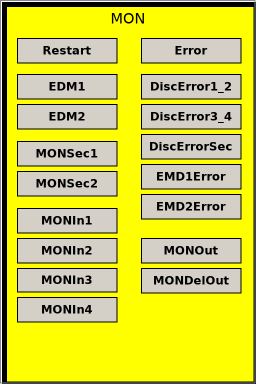
VISUALIZATION V_PH_MON  // 256x384
VAR_INPUT
	stSafetyMon				: ST_SAFETY_FBMON;
	
END_VAR
    Rectangle (2,2 256x384), colour toggle: stSafetyMon.bGeneralError
    Label (5,6 246x25), "MON"
    RoundedRectangle (17,38 100x25), "Restart", colour toggle: stSafetyMon.uStatus.stStatusWords.wInputs.0
    RoundedRectangle (17,74 100x25), "EDM1", colour toggle: stSafetyMon.uStatus.stStatusWords.wInputs.1
    RoundedRectangle (17,297 100x25), "MONIn4", colour toggle: stSafetyMon.uStatus.stStatusWords.wInputs.11
    RoundedRectangle (17,104 100x25), "EDM2", colour toggle: stSafetyMon.uStatus.stStatusWords.wInputs.2
    RoundedRectangle (17,171 100x25), "MONSec2", colour toggle: stSafetyMon.uStatus.stStatusWords.wInputs.4
    RoundedRectangle (17,268 100x24), "MONIn3", colour toggle: stSafetyMon.uStatus.stStatusWords.wInputs.10
    RoundedRectangle (17,141 100x25), "MONSec1", colour toggle: stSafetyMon.uStatus.stStatusWords.wInputs.3
    RoundedRectangle (17,238 100x25), "MONIn2", colour toggle: stSafetyMon.uStatus.stStatusWords.wInputs.9
    RoundedRectangle (17,208 100x25), "MONIn1", colour toggle: stSafetyMon.uStatus.stStatusWords.wInputs.8
    RoundedRectangle (141,74 100x25), "DiscError1_2", colour toggle: stSafetyMon.uStatus.stStatusWords.wDiagnosis.0, invisible if: NOT stSafetyMon.uStatus.stStatusWords.wDiagnosis.0
    RoundedRectangle (141,104 100x25), "DiscError3_4", colour toggle: stSafetyMon.uStatus.stStatusWords.wDiagnosis.1, invisible if: NOT stSafetyMon.uStatus.stStatusWords.wDiagnosis.1
    RoundedRectangle (141,134 100x25), "DiscErrorSec", colour toggle: stSafetyMon.uStatus.stStatusWords.wDiagnosis.2, invisible if: NOT stSafetyMon.uStatus.stStatusWords.wDiagnosis.2
    RoundedRectangle (141,194 100x25), "EMD2Error", colour toggle: stSafetyMon.uStatus.stStatusWords.wDiagnosis.5, invisible if: NOT stSafetyMon.uStatus.stStatusWords.wDiagnosis.5
    RoundedRectangle (141,164 100x25), "EMD1Error", colour toggle: stSafetyMon.uStatus.stStatusWords.wDiagnosis.4, invisible if: NOT stSafetyMon.uStatus.stStatusWords.wDiagnosis.4
    RoundedRectangle (141,38 100x25), "Error", colour toggle: stSafetyMon.uStatus.stStatusWords.wOutputs.0
    RoundedRectangle (141,238 100x25), "MONOut", colour toggle: stSafetyMon.uStatus.stStatusWords.wOutputs.1
    RoundedRectangle (141,268 100x25), "MONDelOut", colour toggle: stSafetyMon.uStatus.stStatusWords.wOutputs.2
    Textfield (17,354 234x25), text list: 'TL_FbState', text index: stSafetyMon.eState
END_VISUALIZATION

(* stored: Version 1.1.0.1, ProductVersion 3.1.4024.4
   Visu V_PH_MON: Id {cdfd986d-dcd7-4418-9435-4fd706e5b2c4} *)
